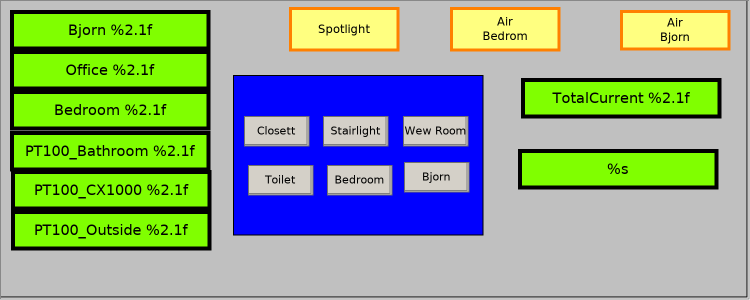
VISUALIZATION TC_VISU  // 750x300
    Rectangle (-3,-3 750x300), text variable: .PCTime
    RoundedRectangle (10,10 200x40), "Bjorn %2.1f", text variable: INT_TO_REAL(.BjornTemp )/10
    RoundedRectangle (10,50 200x40), "Office %2.1f", text variable: INT_TO_REAL (.OfficeTemp) /10
    RoundedRectangle (10,90 200x40), "Bedroom %2.1f", text variable: INT_TO_REAL (.BedRoomTemp) /10
    RoundedRectangle (521,78 200x40), "TotalCurrent %2.1f", text variable: INT_TO_REAL(.TotalCurrent )/10
    RoundedRectangle (620,10 110x40), "Air Bjorn", text variable: AirBjorn, colour toggle: AirBjorn
        toggle AirBjorn
    RoundedRectangle (450,7 110x44), "Air Bedrom", text variable: AirBedroom, colour toggle: AirBedroom
        toggle AirBedroom
    RoundedRectangle (233,75 250x160)
    Button (244,116 65x30), "Closett", text variable: WalkingClosett, colour toggle: WalkingClosett
        toggle WalkingClosett
    Button (323,116 65x30), "Stairlight", text variable: StairLight, colour toggle: StairLight
        toggle StairLight
    Button (403,116 65x30), "Wew Room", colour toggle: Livingroom
        toggle Livingroom p2164770859=TRUE
    Button (248,165 65x30), "Toilet", text variable: ToiletLight, colour toggle: ToiletLight
        toggle ToiletLight
    Button (327,165 65x30), "Bedroom", text variable: BedRoomLight, colour toggle: BedRoomLight
        toggle BedRoomLight
    Button (404,162 65x30), "Bjorn", text variable: BjornLight, colour toggle: BjornLight
        toggle BjornLight
    RoundedRectangle (289,7 110x44), "Spotlight", text variable: SpotLight, colour toggle: SpotLight
        toggle SpotLight
    RoundedRectangle (10,131 200x40), "PT100_Bathroom %2.1f", text variable: INT_TO_REAL(.PT100_Bathroom)/10
        p4168582468: TotalCurrent )/10
    RoundedRectangle (11,170 200x40), "PT100_CX1000 %2.1f", text variable: INT_TO_REAL(PT100_CX1000 )/10
        p4168582468: INT_TO_REAL(.TotalCurrent )/10
    RoundedRectangle (11,210 200x40), "PT100_Outside %2.1f", text variable: INT_TO_REAL(PT100_Outside)/10
    RoundedRectangle (518,149 200x40), "%s", text variable: .RTClock .LokalClock
END_VISUALIZATION

(* stored: Version 1.1.0.1, ProductVersion 3.1.4024.12
   Visu TC_VISU: Id {e13df933-ef21-44f4-8590-64da53a5a79d} *)
